// TIA Portal V19 export
TYPE "LEXCHANGETRAY_typePc_sim"
// stored: Access Published
   STRUCT
      upperNg : Int := 8;   // reandom Ng number
   END_STRUCT;
END_TYPE
